	F1_count: INT;
	F2_count: INT;
	F3_count: INT;
	F4_count: INT;
	F5_count: INT;
	S1_count: INT;
	S2_count: INT;
	R1_count: INT;
	R2_count: INT;
	R3_count: INT;
	R4_count: INT;
	R5_count: INT;
	D1_count: INT;
	C1_count: INT;
	C2_count: INT;
	C3_count: INT;
	U1_count: INT;
	U2_count: INT;
	U3_count: INT;
	radio_count: INT;
	sirena_count: INT;
	allarm_trig: R_TRIG;
	rtrig_radio: R_TRIG;
	rtrig_sirena: R_TRIG;
END_VAR

act();
(*Ritardo avvio allarme su accensione*)
//Timer_allarme(IN:= allarme, PT:= delay_allarme_on, Q=> allarme_on, ET=> );
(*Sensori*)
rilevato_movimento:=
	NOT (	
	SM_F1 AND
	SM_F2 AND
	SM_F3 AND
	SM_F4 AND
	SM_F5 AND
	SM_S1 AND
	SM_S2 AND
	//SM_R1 AND
	//SM_R2 AND
	//SM_R3 AND
	//SM_R4 AND
	//SM_R5 AND
	//SM_D1 AND
	SM_C1 AND
	//SM_C2 AND
	//SM_C3 AND
	SM_U1 AND 
	SM_U2 //AND
	//SM_U3 
	);
(*rilevata_manomissione:=NOT (Tamper_interno AND Tamper_fronte AND Tamper_retro AND Tamper_sinistro);*)
(*Ritardo spegnimento sirena*)
//Timer_Sirena(IN:= timer_Allarme.Q  AND rilevato_movimento, PT:= delay_sirena_off, Q=>, ET=> );
(*Azioni allarme*)
(*Segnale_sirena:=(timer_sirena.Q  AND NOT alarm_service) OR test_sirena;*)
//Segnale_radio:=(timer_sirena.Q AND NOT alarm_service) OR test_radio;
(*Allarme Tamper*)
allarme_tamper:=NOT alarm_service AND rilevata_manomissione;

IF allarme_Attivo<>0 (*allarme_on*) THEN
	//Gestione contatore sensore F1
	F1_trig(CLK:= SM_F1, Q=> );
	IF F1_trig.Q THEN
		F1_count:=F1_count+1;
	END_IF
	//Gestione contatore sensore F2
	F2_trig(CLK:= SM_F2, Q=> );
	IF F2_trig.Q THEN
		F2_count:=F2_count+1;
	END_IF
	//Gestione contatore sensore F3
	F3_trig(CLK:= SM_F3, Q=> );
	IF F3_trig.Q THEN
		F3_count:=F3_count+1;
	END_IF
	//Gestione contatore sensore F4
	F4_trig(CLK:= SM_F4, Q=> );
	IF F4_trig.Q THEN
		F4_count:=F4_count+1;
	END_IF
	//Gestione contatore sensore F5
	F5_trig(CLK:= SM_F5, Q=> );
	IF F5_trig.Q THEN
		F5_count:=F5_count+1;
	END_IF
	//Gestione contatore sensore S1
	S1_trig(CLK:= SM_S1, Q=> );
	IF S1_trig.Q THEN
		S1_count:=S1_count+1;
	END_IF
	//Gestione contatore sensore S2
	S2_trig(CLK:= SM_S2, Q=> );
	IF S2_trig.Q THEN
		S2_count:=S2_count+1;
	END_IF
	(*//Gestione contatore sensore R1
	R1_trig(CLK:= SM_R1, Q=> );
	IF R1_trig.Q THEN
		R1_count:=R1_count+1;
	END_IF
	//Gestione contatore sensore R2
	R2_trig(CLK:= SM_R2, Q=> );
	IF R2_trig.Q THEN
		R2_count:=R2_count+1;
	END_IF
	//Gestione contatore sensore R3
	R3_trig(CLK:= SM_R3, Q=> );
	IF R3_trig.Q THEN
		R3_count:=R3_count+1;
	END_IF
	//Gestione contatore sensore R4
	R4_trig(CLK:= SM_R4, Q=> );
	IF R4_trig.Q THEN
		R4_count:=R4_count+1;
	END_IF
	//Gestione contatore sensore R5
	R5_trig(CLK:= SM_R5, Q=> );
	IF R5_trig.Q THEN
		R5_count:=R5_count+1;
	END_IF
	//Gestione contatore sensore D1
	D1_trig(CLK:= SM_D1, Q=> );
	IF D1_trig.Q THEN
		D1_count:=D1_count+1;
	END_IF*)
	//Gestione contatore sensore C1
	C1_trig(CLK:= SM_C1, Q=> );
	IF C1_trig.Q THEN
		C1_count:=C1_count+1;
	END_IF
	(*//Gestione contatore sensore C2
	C2_trig(CLK:= SM_C2, Q=> );
	IF C2_trig.Q THEN
		C2_count:=C2_count+1;
	END_IF
	//Gestione contatore sensore C3
	C3_trig(CLK:= SM_C3, Q=> );
	IF C3_trig.Q THEN
		C3_count:=C3_count+1;
	END_IF*)
	//Gestione contatore sensore U1
	U1_trig(CLK:= SM_U1, Q=> );
	IF U1_trig.Q THEN
		U1_count:=U1_count+1;
	END_IF
	//Gestione contatore sensore U2
	U2_trig(CLK:= SM_U2, Q=> );
	IF U2_trig.Q THEN
		U2_count:=U2_count+1;
	END_IF
	(*//Gestione contatore sensore U3
	U3_trig(CLK:= SM_U3, Q=> );
	IF U3_trig.Q THEN
		U3_count:=U3_count+1;
	END_IF*)
	//Gestione contatore segnale radio e sirena
	rtrig_radio(CLK:= segnale_radio, Q=> );
	rtrig_sirena(CLK:= segnale_sirena, Q=> );
	IF rtrig_radio.Q THEN
		radio_count:=radio_count+1;
	END_IF
	IF rtrig_sirena.Q THEN
		sirena_count:=sirena_count+1;
	END_IF
END_IF
allarm_trig(CLK:= allarme_Attivo<>0 (*allarme*), Q=> );
IF allarm_trig.Q THEN
	F1_count:=0;
	F2_count:=0;
	F3_count:=0;
	F4_count:=0;
	F5_count:=0;
	S1_count:=0;
	S2_count:=0;
	R1_count:=0;
	R2_count:=0;
	R3_count:=0;
	R4_count:=0;
	R5_count:=0;
	D1_count:=0;
	C1_count:=0;
	C2_count:=0;
	C3_count:=0;
	U1_count:=0;
	U2_count:=0;
	U3_count:=0;
	radio_count:=0;
	sirena_count:=0;
END_IF
//Gestione sensori movimento
sensori_STRU[0](indice:=0); //Sensore movimento frontale 1
sensori_STRU[1](indice:=1); //Sensore movimento frontale 2
sensori_STRU[2](indice:=2); //Sensore movimento frontale 3
sensori_STRU[3](indice:=3); //Sensore movimento frontale 4
sensori_STRU[4](indice:=4); //Sensore movimento frontale 5
sensori_STRU[5](indice:=5); //Sensore movimento sinistro 1
sensori_STRU[6](indice:=6); //Sensore movimento sinistro 2
sensori_STRU[7](indice:=7); //Sensore movimento retro 1
sensori_STRU[8](indice:=8); //Sensore movimento retro 2
sensori_STRU[9](indice:=9); //Sensore movimento retro 3
sensori_STRU[10](indice:=10); //Sensore movimento retro 4
sensori_STRU[11](indice:=11); //Sensore movimento retro 5
sensori_STRU[12](indice:=12); //Sensore movimento destro
sensori_STRU[13](indice:=13); //Sensore movimento centrale 1
sensori_STRU[14](indice:=14); //Sensore movimento centrale 2
sensori_STRU[15](indice:=15); //Sensore movimento centrale 3
sensori_STRU[16](indice:=16); //Sensore movimento ufficio tecnico U1
sensori_STRU[17](indice:=17); //Sensore movimento locale svago U2
sensori_STRU[18](indice:=18); //Sensore movimento ingresso U3

//Attivazione segnale sirena-radio allarme
IF ((sens_allarme_Stru[0].allarme_sensore OR 
	sens_allarme_stru[1].allarme_sensore OR
	sens_allarme_Stru[2].allarme_sensore OR
	sens_allarme_stru[3].allarme_sensore OR
	sens_Allarme_stru[4].allarme_sensore OR
	sens_allarme_stru[5].allarme_sensore OR
	sens_allarme_Stru[6].allarme_sensore OR
	sens_allarme_stru[13].allarme_sensore OR
	sens_allarme_Stru[16].allarme_sensore OR
	sens_allarme_Stru[17].allarme_sensore) AND NOT alarm_Service) THEN
		allarme_scattato:=TRUE;
ELSE
		allarme_scattato:=FALSE;
END_IF
segnale_sirena:=(allarme_Scattato AND HMI_sirena) OR test_sirena;	
segnale_radio:=(allarme_scattato AND HMI_radio) OR test_radio;
ingresso_sens[0]:=SM_F1;
ingresso_sens[1]:=SM_F2;
ingresso_sens[2]:=SM_F3;
ingresso_sens[3]:=SM_F4;
ingresso_sens[4]:=SM_F5;
ingresso_sens[5]:=SM_S1;
ingresso_sens[6]:=SM_S2;
ingresso_sens[13]:=SM_C1;
ingresso_sens[16]:=SM_U1;
ingresso_sens[17]:=SM_U2;

ACTION ACT:
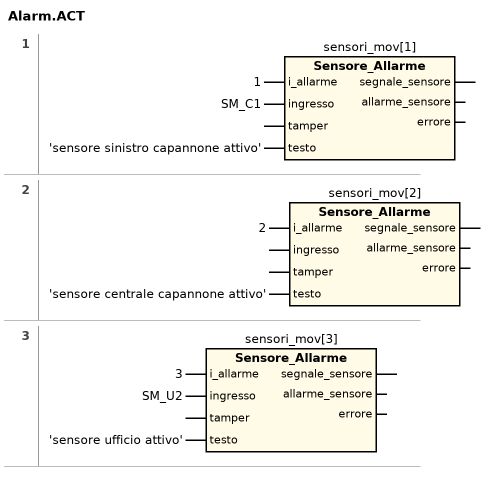
// NETWORK 1
sensori_mov[1](i_allarme := 1, ingresso := SM_C1, testo := 'sensore sinistro capannone attivo'); // Sensore_Allarme

// NETWORK 2
sensori_mov[2](i_allarme := 2, testo := 'sensore centrale capannone attivo'); // Sensore_Allarme

// NETWORK 3
sensori_mov[3](i_allarme := 3, ingresso := SM_U2, testo := 'sensore ufficio attivo'); // Sensore_Allarme
END_ACTION

END_PROGRAM

// ---- POUs/ProjetcFB/Sensore_Allarme.TcPOU
FUNCTION_BLOCK Sensore_Allarme
VAR_INPUT
	i_allarme: INT;
	ingresso: BOOL; // segnale fisico sensore BOOL
	tamper: BOOL;
	testo: STRING;
END_VAR
VAR_OUTPUT
	segnale_sensore: BOOL;
	allarme_sensore: BOOL;
	errore: BYTE; //0=OK-1=allarme attivo-2=dispositivo aperto-3=movimento diffettoso-4=tamper
END_VAR
VAR
	delay_on: TON;
	a1: BOOL;
	timer_sendif: TON;//timer per rilevamento sensore difettoso
	sensore: BOOL;
	pulse_sensor: TP;
	
	x: INT:=1; //Indice per testo allarmi
	trig_ingresso: F_TRIG;
	ufficio1: F_TRIG;
	ufficio2: F_TRIG;
	ufficio3: F_TRIG;
	capannone: F_TRIG;
END_VAR

pulse_sensor(IN:=ingresso , PT:=T#1S , Q=>sensore , ET=> );
sens_allarme[i_allarme].sens_mov:=TRUE;
IF sens_allarme[i_allarme].sens_attivo THEN
	IF (mode_a=0 AND sens_allarme[i_allarme].mode_a0) OR 
		(mode_a=1 AND sens_allarme[i_allarme].mode_a1) OR
		(mode_a=2 AND sens_allarme[i_allarme].mode_a2) OR
		(mode_a=3 AND sens_allarme[i_allarme].mode_a3) OR
		(mode_a=4 AND sens_allarme[i_allarme].mode_a4) THEN
		IF sens_allarme[i_allarme].sens_ritardato THEN
			delay_on(IN:= NOT sensore AND allarme_on, PT:= sens_allarme[i_allarme].delay_allarme, Q=> , ET=> );
		ELSE
			a1:=NOT sensore AND allarme_on;	
		END_IF
	allarme_sensore:=a1 OR delay_on.Q;
	END_IF
END_IF
timer_sendif(IN:= NOT sensore AND allarme_on, PT:= T#1H, Q=> , ET=> );
IF sensore THEN
	errore:=0;
ELSIF allarme_sensore THEN
	errore:=1;
ELSIF sens_allarme[i_allarme].porta_fin AND NOT sensore THEN
	errore:=2;
ELSIF NOT sens_allarme[i_allarme].porta_fin AND timer_sendif.Q  THEN
	errore:=3;
ELSIF NOT tamper THEN
	errore:=4;
END_IF

END_FUNCTION_BLOCK

// ---- POUs/Timbrature.TcPOU
PROGRAM Timbrature
VAR
	puls_timbro: BOOL;
	stringa_2: STRING;
	stringa:STRING(23);
	i:STRING;
	Tempo_scrittura: TP;
	Tempo_chiusura: TP;
	chiudi: BOOL;
	Scrivi_action: F_TRIG;
	Chiudi_action:F_TRIG;
	anno: STRING;
	
	i_utente_su: R_TRIG;
	i_utente_giu: R_TRIG;
	save_par_all: R_TRIG;
	
	stampa_report: NT_StartProcess;
	HMI_stampa: BOOL;
END_VAR

//Creazione stringa per file di testo
anno:=word_to_decstr(ora_plc.TIMESTR.wYear-2000,2);
IF ekey_scanner_produzione.bGoodFinger THEN
	stringa:=concat(stringa,'01');
	stringa:=concat(stringa,WORD_TO_DECSTR(ora_plc.TIMESTR.wMonth,2));
	stringa:=concat(stringa,WORD_TO_DECSTR(ora_plc.TIMESTR.wDay,2));
	stringa:=concat(stringa,WORD_TO_DECSTR(ora_plc.TIMESTR.wHour,2));
	stringa:=concat(stringa,WORD_TO_DECSTR(ora_plc.TIMESTR.wMinute,2));
	stringa:=concat(stringa,utenti[ekey_scanner_produzione.byRecUserID].num_badge);
	stringa:=concat(stringa,'0000E');
	stringa:=concat(stringa,anno);
	stringa_2:=stringa;
	stringa:='';
END_IF
//Apertura file di testo
apri_file(
	sNetId:= , 
	sPathName:= 'C:\timbrature\Datafil.txt', 
	nMode:= FOPEN_MODEAPPEND, 
	ePath:= , 
	bExecute:= ekey_scanner_produzione.bGoodFinger AND NOT hmi_finger AND NOT hmi_finger_RFID,
	tTimeout:= , 
	bBusy=> , 
	bError=> , 
	nErrId=> , 
	hFile=> );
Tempo_scrittura(IN:= ekey_scanner_produzione.bGoodFinger, PT:=T#1S , Q=> , ET=> );
//Inserimento orari nel file di testo
Scrivi_action(CLK:=tempo_scrittura.Q , Q=> );
inserisci_testo(
	sNetId:= , 
	hFile:= apri_file.hFile, 
	sLine:= concat(stringa_2,'$R$N'), 
	bExecute:= scrivi_action.Q, 
	tTimeout:= , 
	bBusy=> , 
	bError=> , 
	nErrId=> );
Tempo_chiusura(IN:= scrivi_action.Q, PT:= T#1S, Q=> , ET=> );

//Chiusura file di testo
Chiudi_action(CLK:=tempo_chiusura.Q , Q=> );
chiudi_file(
	sNetId:= , 
	hFile:= apri_file.hFile, 
	bExecute:= chiudi_action.Q OR chiudi, 
	tTimeout:= , 
	bBusy=> , 	
	bError=> , 
	nErrId=> );
	
//Gestione utenti su HMI
i_utente_su(CLK:= hmi_utentesu , Q=> );
i_utente_giu(CLK:= hmi_utentegiu , Q=> );
IF i_utente_su.Q AND indice_utente<Nmu THEN
	indice_utente:= indice_utente+1;
END_IF
IF i_utente_giu.Q AND indice_utente>1 THEN
	indice_utente:= indice_utente-1;
END_IF
IF i_utente_giu.Q OR i_utente_su.Q OR HMI_annulla THEN
	HMI_user_type:= utenti[indice_utente].user_type;
	HMI_num_badge:= utenti[indice_utente].num_badge;
	HMI_nome_utente:= utenti[indice_utente].nome_utente;
END_IF;
save_par_all(CLK:= HMI_save_utente, Q=> );
IF save_par_all.Q THEN
	utenti[indice_utente].user_type:= HMI_user_type;
	utenti[indice_utente].num_badge:= HMI_num_badge;
	utenti[indice_utente].nome_utente:= HMI_nome_utente;
END_IF

stampa_report(
	NETID:= , 
	PATHSTR:= 'powershell.exe', 
	DIRNAME:= , 
	COMNDLINE:= 'Get-Content c:\prova.txt | Out-Printer', 
	START:= HMI_stampa, 
	TMOUT:= T#5S, 
	BUSY=> , 
	ERR=> , 
	ERRID=> );

END_PROGRAM

// ---- POUs/ProjetcFB/Sensore_Allarme_STRU.TcPOU
FUNCTION_BLOCK Sensore_Allarme_STRU
VAR_INPUT
	indice:BYTE;
END_VAR
VAR
	pulse_sensore: TP; //Tempo impulso suono sirena
	trig_sensore: F_TRIG;
	Ritardo_Off_Sens: TON; //Ritardo spegnimento sensore
	att_ritardo_off: BOOL; //Attivazione timer ritardo spegnimento sensore
	SR_tamper: SR;
	Ritardo_inserimento: TON;
END_VAR

//Conversione tempi ritardi da INT a TIME
sens_allarme_stru[indice].ritardo_ON:=REAL_TO_TIME(sens_allarme_stru[indice].HMI_Ritardo_ON*1000);
sens_allarme_stru[indice].ritardo_OFF:=REAL_TO_TIME(sens_allarme_stru[indice].HMI_Ritardo_OFF*1000);
//Ritardo attivazione sensore
Ritardo_inserimento(IN:= allarme_attivo<>0, PT:= sens_allarme_stru[indice].ritardo_ON, Q=> , ET=> );

IF sens_allarme_stru[indice].sens_ON_OFF AND Ritardo_inserimento.Q THEN
	IF 	(allarme_Attivo=1 AND sens_allarme_stru[indice].sens_zonaA) OR
		(allarme_attivo=2 AND sens_allarme_stru[indice].sens_zonaB) OR
		(allarme_attivo=3 AND sens_allarme_stru[indice].sens_zonaC) OR
		(allarme_Attivo=4 AND sens_allarme_stru[indice].sens_zonaD) THEN
		trig_sensore(CLK:= ingresso_sens[indice], Q=> );
		IF trig_sensore.Q THEN
			att_ritardo_off:=TRUE;
			sens_allarme_stru[indice].sensore_preallarme:=TRUE;
		END_IF
		Ritardo_Off_Sens(IN:= att_ritardo_off, PT:= sens_allarme_stru[indice].ritardo_off, Q=> , ET=> );
		pulse_sensore(IN:= ritardo_off_sens.Q, PT:= T#1M, Q=> sens_allarme_stru[indice].allarme_sensore, ET=> );
	END_IF
END_IF

IF allarme_Attivo=0 THEN
	sens_allarme_stru[indice].allarme_sensore:=FALSE;
	att_ritardo_off:=FALSE;
	sens_allarme_stru[indice].sensore_preallarme:=FALSE;
END_IF
//Reset allarme sensore
IF reset_Allarme THEN
	sens_allarme_stru[indice].allarme_sensore:=FALSE;
END_IF
//Gestione tamper sensore
SR_tamper(SET1:= NOT tamper[indice], RESET:= reset_tamper, Q1=> sens_allarme_stru[indice].tamper_sensore);
//Designazione bit di stato sensore
IF NOT sens_allarme_stru[indice].sens_ON_OFF THEN
	sens_allarme_stru[indice].stato_sensore:=0;
ELSIF sens_allarme_stru[indice].sens_ON_OFF AND sens_allarme_stru[indice].allarme_sensore THEN
	sens_allarme_stru[indice].stato_sensore:=1;
ELSIF NOT tamper[indice] THEN
	sens_allarme_stru[indice].stato_sensore:=2;
ELSIF 	sens_allarme_stru[indice].sens_ON_OFF AND
		((allarme_attivo=1 AND sens_allarme_stru[indice].sens_zonaA) OR
		(allarme_attivo=2 AND sens_allarme_stru[indice].sens_zonaB) OR
		(allarme_Attivo=3 AND sens_allarme_stru[indice].sens_zonaC) OR
		(allarme_attivo=4 AND sens_allarme_stru[indice].sens_zonaD)) AND NOT ingresso_sens[indice] THEN
	sens_allarme_stru[indice].stato_sensore:=3;
ELSIF 	sens_allarme_stru[indice].sens_ON_OFF AND
		((allarme_attivo=1 AND sens_allarme_stru[indice].sens_zonaA) OR
		(Allarme_attivo=2 AND sens_allarme_stru[indice].sens_zonaB) OR
		(Allarme_attivo=3 AND sens_allarme_stru[indice].sens_zonaC) OR
		(Allarme_attivo=4 AND sens_allarme_stru[indice].sens_zonaD)) AND ingresso_sens[indice] THEN
	sens_allarme_stru[indice].stato_sensore:=4;
ELSIF sens_allarme_stru[indice].sens_ON_OFF AND ingresso_sens[indice] THEN
	sens_allarme_stru[indice].stato_sensore:=5;
ELSIF sens_allarme_stru[indice].sens_ON_OFF AND NOT ingresso_sens[indice] THEN
	sens_allarme_stru[indice].stato_sensore:=6;
END_IF
//Gestione manutenzione sensore
IF manutenzione_sensore THEN
	sens_allarme_stru[indice].sens_ON_OFF:=FALSE;
END_IF

END_FUNCTION_BLOCK

// ---- POUs/ADS_CX8080.TcPOU
PROGRAM ADS_CX8080
VAR
	ADS_read: ADSREAD;
	ADS_Write: ADSWRITE;
END_VAR

//Lettura variabili da modulo CX8080 con ADS
ADS_read(
	NETID:= '5.41.109.126.1.1', //AmsnetID del secondo PLC
	PORT:= 801, 
	IDXGRP:=16#4020 , 
	IDXOFFS:=2000 , 
	LEN:= SIZEOF(segnalird), 
	DESTADDR:= ADR(segnalird), 
	READ:= aggiorna=1, 
	TMOUT:=T#5S, 
	BUSY=> , 
	ERR=> , 
	ERRID=> );
//Scrittura variabili su modulo CX8080 con ADS
ADS_Write(
	NETID:= '5.41.109.126.1.1', //AmsnetID del secondo PLC
	PORT:= 801, 
	IDXGRP:= 16#4020, 
	IDXOFFS:= 1000, 
	LEN:= SIZEOF(segnaliwr), 
	SRCADDR:= ADR(segnaliwr), 
	WRITE:= aggiorna=1, 
	TMOUT:=T#5S , 
	BUSY=> , 
	ERR=> , 
	ERRID=> );

END_PROGRAM

// ---- POUs/ProjetcFB/DALI_TK_SR07.TcPOU
FUNCTION_BLOCK DALI_TK_SR07
VAR_INPUT
	ID : DWORD;
END_VAR
VAR_OUTPUT
	Temp : UINT; (*Valore * 10 - 10,0°C => 100*)
END_VAR
VAR
	READ: FB_Rec_Generic;
	temperatura: DINT;
END_VAR

READ(
	str_KL6581:=enocean_buffer , 
	byNode:=1 , 
	dw_ID:=ID , 
	ar_Value=> , 
	by_Node=> , 
	by_STATE=> , 
	bReceive=> , 
	EnOceanTyp=> );
temperatura:=TRUNC((255-read.ar_Value[1])/0.6375);	
temp:=DINT_TO_UINT (temperatura);

END_FUNCTION_BLOCK
